FUNCTION_BLOCK DrillStation_FORTEInterface (* Basic Function Block Type *)
  (* Standard: 61499-2 *)
  (* Version 0.2, 2003-12-04, JHC, Rockwell Automation, Renamed for better indexing. *)
  (* Version 0.1, 2002-11-05, JHC, Rockwell Automation, Corrected missing ST element in Algorithm REQ. *)
  (* Version 0.0, 2000-05-30, JHC, Rockwell Automation *)
  (* Compiler header: package fb.rt.benchmarks.DrillStation; *)
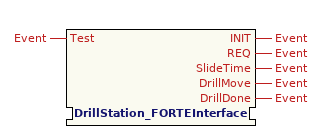
  EVENT_INPUT
    Test; (* Initialization Request *)
  END_EVENT
  EVENT_OUTPUT
    INIT; (* Initialization Request *)
    REQ; (* Normal Execution Request *)
    SlideTime;
    DrillMove;
    DrillDone;
  END_EVENT
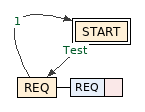
  EC_STATES
    START; (* Initial State *)
    REQ : REQ; (* Normal execution *)
  END_STATES
  EC_TRANSITIONS
    START TO REQ := Test;
    REQ TO START := 1;
  END_TRANSITIONS
  ALGORITHM REQ IN ST: (* Normally executed algorithm *)
(*
File Code goes here
*)
  END_ALGORITHM
END_FUNCTION_BLOCK
